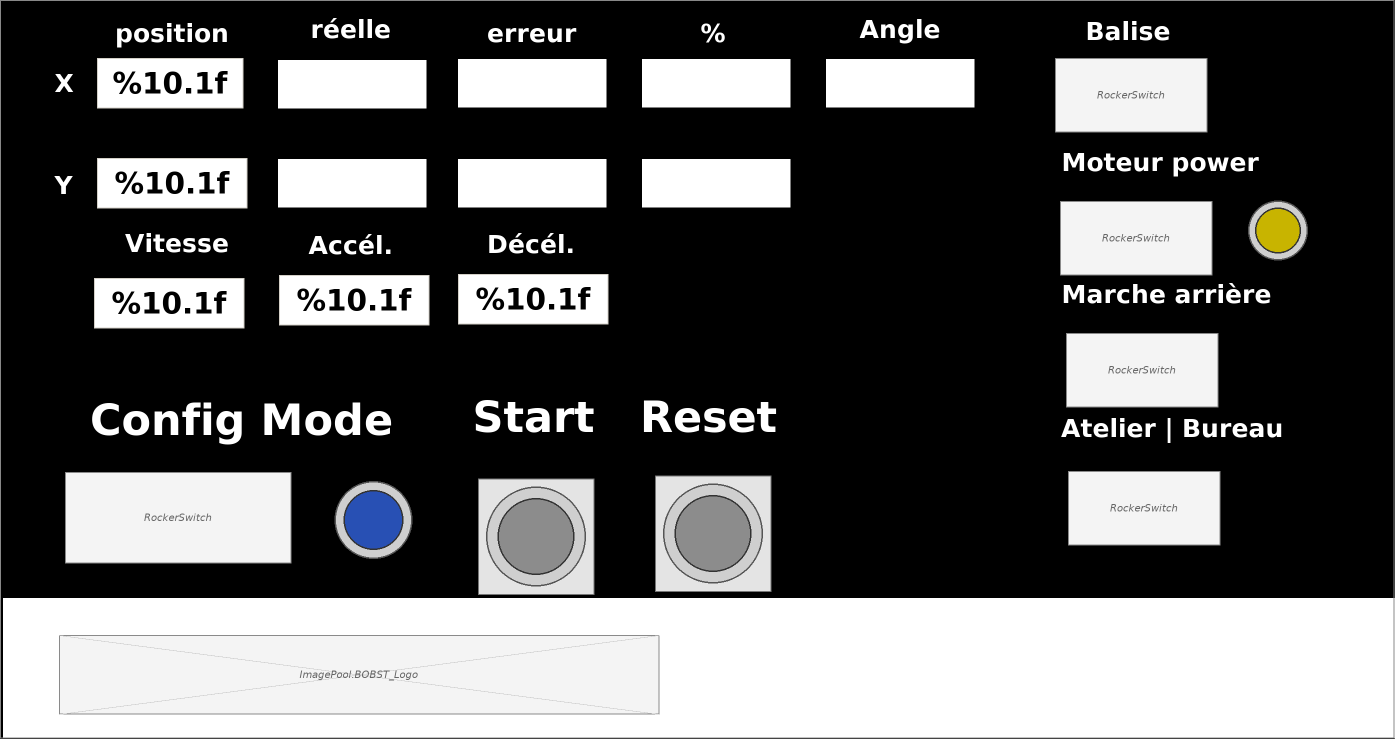
VISUALIZATION V_Config  // 1395x739
    Rectangle (3,598 1396x140)
    Rectangle (457,158 150x50), "%10.1f", text variable: G_Visus.lrConfigErreurY
    Label (97,8 150x50), "position"
    Label (276,4 150x50), "réelle"
    Label (457,8 150x50), "erreur"
    Label (663,8 100x50), "%"
    Textfield (97,58 146x50), "%10.1f", text variable: G_Visus.lrConfigPosX
        OnMouseDown: write G_Visus.lrConfigPosX via InputWithLimits, min 0, max 1000000
    Textfield (97,158 150x50), "%10.1f", text variable: G_Visus.lrConfigPosY
        OnMouseDown: write G_Visus.lrConfigPosY via InputWithLimits, min 0, max 3000
    Rectangle (277,59 150x50), "%10.1f", text variable: G_Odometrie.lrPositionX
    Rectangle (277,158 150x50), "%10.1f", text variable: G_Odometrie.lrPositionY
    Rectangle (457,58 150x50), "%10.1f", text variable: G_Visus.lrConfigErreurX
    Rectangle (641,58 150x50), "%10.1f", text variable: G_Visus.lrConfigErreurX_Pourcent
    Rectangle (641,158 150x50), "%10.1f", text variable: G_Visus.lrConfigErreurY_pourcent
    Label (40,58 49x50), "X"
    Label (39,160 49x50), "Y"
    Rectangle (825,58 150x50), "%10.1f", text variable: G_Odometrie.lrAngleDeg
    Label (825,4 150x50), "Angle"
    Textfield (94,278 150x50), "%10.1f", text variable: G_Visus.lrConfigVitesse
        OnMouseDown: write G_Visus.lrConfigVitesse via InputWithLimits, min 0, max 1700
    Label (102,218 150x50), "Vitesse"
    Label (258,220 186x50), "Accél."
    Label (429,219 204x50), "Décél."
    Textfield (279,275 150x50), "%10.1f", text variable: G_Visus.lrConfigAcc
        OnMouseDown: write G_Visus.lrConfigAcc via Default, min 0, max 1500
    Textfield (458,274 150x50), "%10.1f", text variable: G_Visus.lrConfigDecc
        OnMouseDown: write G_Visus.lrConfigDecc via InputWithLimits, min 0, max 1500
    RockerSwitch (1055,58 152x74), variable: G_Visus.bConfigBalise, behaviour: TOGGLE, style: Switch-RockerSwitch-Gray
    Label (1053,6 150x50), "Balise"
    RockerSwitch (65,472 226x91), variable: G_Visus.bConfigEnable, behaviour: TOGGLE, style: Switch-RockerSwitch-Gray
    Label (72,392 339x56), "Config Mode"
    Lamp1 (322,475 103x90), variable: G_Visus.bConfigReady, style: Lamp-Lamp1-Blue
    RockerSwitch (1060,201 152x74), variable: G_Visus.bConfigMoteurPower, behaviour: TOGGLE, style: Switch-RockerSwitch-Gray
    Label (1059,137 203x50), "Moteur power"
    Lamp1 (1242,196 72x69), variable: G_Visus.bConfigMoteurReady, style: Lamp-Lamp1-Yellow
    RockerSwitch (1066,333 152x74), variable: G_Visus.bConfigMarcheArriere, behaviour: TOGGLE, style: Switch-RockerSwitch-Gray
    Label (1065,269 203x50), "Marche arrière"
    PushSwitch (478,466 116x141), variable: G_Visus.bConfigStart, behaviour: TOGGLE, style: Switch-PushSwitch-Gray
    Label (447,392 173x50), "Start"
    PushSwitch (655,463 116x141), variable: G_Visus.bConfigReset, behaviour: TAP, style: Switch-PushSwitch-Gray
    Label (625,392 167x50), "Reset"
    Label (1064,403 217x50), "Atelier | Bureau"
    RockerSwitch (1068,471 152x74), variable: G_Visus.bConfigChoixCote, behaviour: TOGGLE, style: Switch-RockerSwitch-Gray
    Image (59,635 600x79), image: ImagePool.BOBST_Logo
        OnMouseDown: change screen: V_Menu
END_VISUALIZATION

(* stored: Version 1.1.0.1, ProductVersion 3.1.4024.11
   Visu V_Config: Id {cd018ebc-9d6e-4dec-b8e6-86ec25903a8e} *)
